// Mitsubishi GX Works2 project: PLC (21)   PLC: FX3G
// PLC

// global labels: Global1
VAR_GLOBAL
  light1 AT Y010 : BOOL;
  EmergencySwitch AT X007 : BOOL;
  OrangeReg AT D1100 : REAL;  (* STARTDAY *)
  TangerineReg AT D1105 : REAL;  (* STARTDAY *)
  PomelaReg AT D1110 : REAL;  (* STARTDAY *)
  OrangeCont AT D1115 : REAL;
  TangerineCont AT D1120 : REAL;
  PomelaCont AT D1125 : REAL;
  startSwitch AT X010 : BOOL;  (* STARTDAY *)
  light2 AT M0 : BOOL;  (* STARTDAY *)
END_VAR
VAR_GLOBAL CONSTANT
  two : REAL := 2;
END_VAR
VAR_GLOBAL
  light3 AT M1 : BOOL;  (* STARTDAY *)
  washSwitch AT X002 : BOOL;
  washTimer AT TC1 : BOOL;
END_VAR
VAR_GLOBAL CONSTANT
  three : INT := 30;
END_VAR
VAR_GLOBAL
  washing AT TS1 : BOOL;
  washLight AT Y005 : BOOL;
END_VAR
VAR_GLOBAL CONSTANT
  countTo3 : INT := 30;  (* שלוש שניות *)
  hundred : REAL := 100;
END_VAR
VAR_GLOBAL
  OrangeWashReg AT D1130 : REAL;
  light4 AT M2 : BOOL;  (* אם יש מעל 100 קג תפוזים *)
END_VAR
VAR_GLOBAL CONSTANT
  zeroConst : REAL;
END_VAR
VAR_GLOBAL
  light5 AT M3 : BOOL;  (* אם יש מתחת ל100 קג תפוזים *)
  light6 AT M4 : BOOL;  (* תפוזים נשטפו *)
END_VAR
VAR_GLOBAL CONSTANT
  half : REAL := 0.5;
END_VAR
VAR_GLOBAL
  PomelaWashReg AT D1135 : REAL;
  TangerineWashReg AT D1140 : REAL;
  light7 AT M5 : BOOL;  (* הכל נשטף *)
  squeezeSwitch AT X001 : BOOL;  (* stage 2 start *)
  squeezeCont AT D1145 : REAL;  (* מיכל סחיטה של כלל הפירות *)
  stage2light AT Y001 : BOOL;
  stage3Switch AT X011 : BOOL;
  stage3Counter AT CC0 : BOOL;
END_VAR
VAR_GLOBAL CONSTANT
  countTo2 : INT := 2;  (* שתי לחיצות *)
END_VAR
VAR_GLOBAL
  stage3Start AT CS0 : BOOL;
  light8 AT M6 : BOOL;
END_VAR
VAR_GLOBAL CONSTANT
  halfSec : INT := 5;
END_VAR
VAR_GLOBAL
  squeezeTimer AT TC2 : BOOL;
  flashing AT TS2 : BOOL;
  flashlight2 AT Y002 : BOOL;
  squeezeTimer2 AT TC3 : BOOL;
  flashlight3 AT Y003 : BOOL;
  flashing2 AT TS3 : BOOL;
  stage3TotalTime AT TC4 : BOOL;
  threeSecOff AT TS4 : BOOL;  (* כיבוי אורות מהבהבים לאחר 3 שניות *)
  light9 AT M7 : BOOL;  (* תהליך הסחיטה הסתיים *)
  juiceCont AT D1150 : REAL;  (* מיכל מיץ סחוט *)
  light10 AT M8 : BOOL;
  analog2 AT D8281 : WORD;
  analogOutput2 AT D1160 : WORD;
END_VAR
VAR_GLOBAL CONSTANT
  fourHundred : REAL := 400.0;
END_VAR
VAR_GLOBAL
  qualityCheckReg AT D1155 : REAL;
END_VAR
VAR_GLOBAL CONSTANT
  One : REAL := 1.0;
  five : REAL := 5.0;
END_VAR
VAR_GLOBAL
  light11 AT M9 : BOOL;
  light12 AT M10 : BOOL;
  qualityIsGood AT Y004 : BOOL;
  qualityIsAmazing AT Y004 : BOOL;
END_VAR
VAR_GLOBAL CONSTANT
  countTo5 : INT := 50;
END_VAR
VAR_GLOBAL
  qualityTimer AT TC5 : BOOL;
  TS05 AT TS5 : BOOL;
  light13 AT M11 : BOOL;
  failCounter AT CC1 : BOOL;
  disgustingJuice AT CS1 : BOOL;  (* נכשל פעמיים בבדיקת איכות *)
  PerfectJuiceStorage AT D1165 : REAL;
  stage4Switch AT X003 : BOOL;
  light14 AT M12 : BOOL;
  light15 AT M13 : BOOL;
  light16 AT M14 : BOOL;
  repairMachine AT X006 : BOOL;  (* התקשרות לטכנאי לתיקון *)
  maxFruitReg AT D1170 : REAL;
  analogOutput AT D8282 : WORD;
  endOfDay AT M15 : BOOL;
  repairTimer AT TC6 : BOOL;  (* זמן תיקון *)
  repairFlash AT TC7 : BOOL;
  repairLight AT Y006 : BOOL;
  light17 AT M16 : BOOL;
  repairFlashING AT TS7 : BOOL;
  repairFakeFlash AT TC8 : BOOL;
  light18 AT M17 : BOOL;
  repairSchedule AT TS8 : BOOL;
  light19 AT M18 : BOOL;
  endOfIteration AT M19 : BOOL;  (* סוף איטרציה *)
  howLongRepair AT D1175 : WORD;
END_VAR

// task Task_01 (event TRUE, interval 0, priority 31): POU_01

PROGRAM POU_01
(* structured ladder/FBD written out as ST: instructions are called as NAME(EN, inputs, outputs); _pN, _eN, _tN stand for wires *)
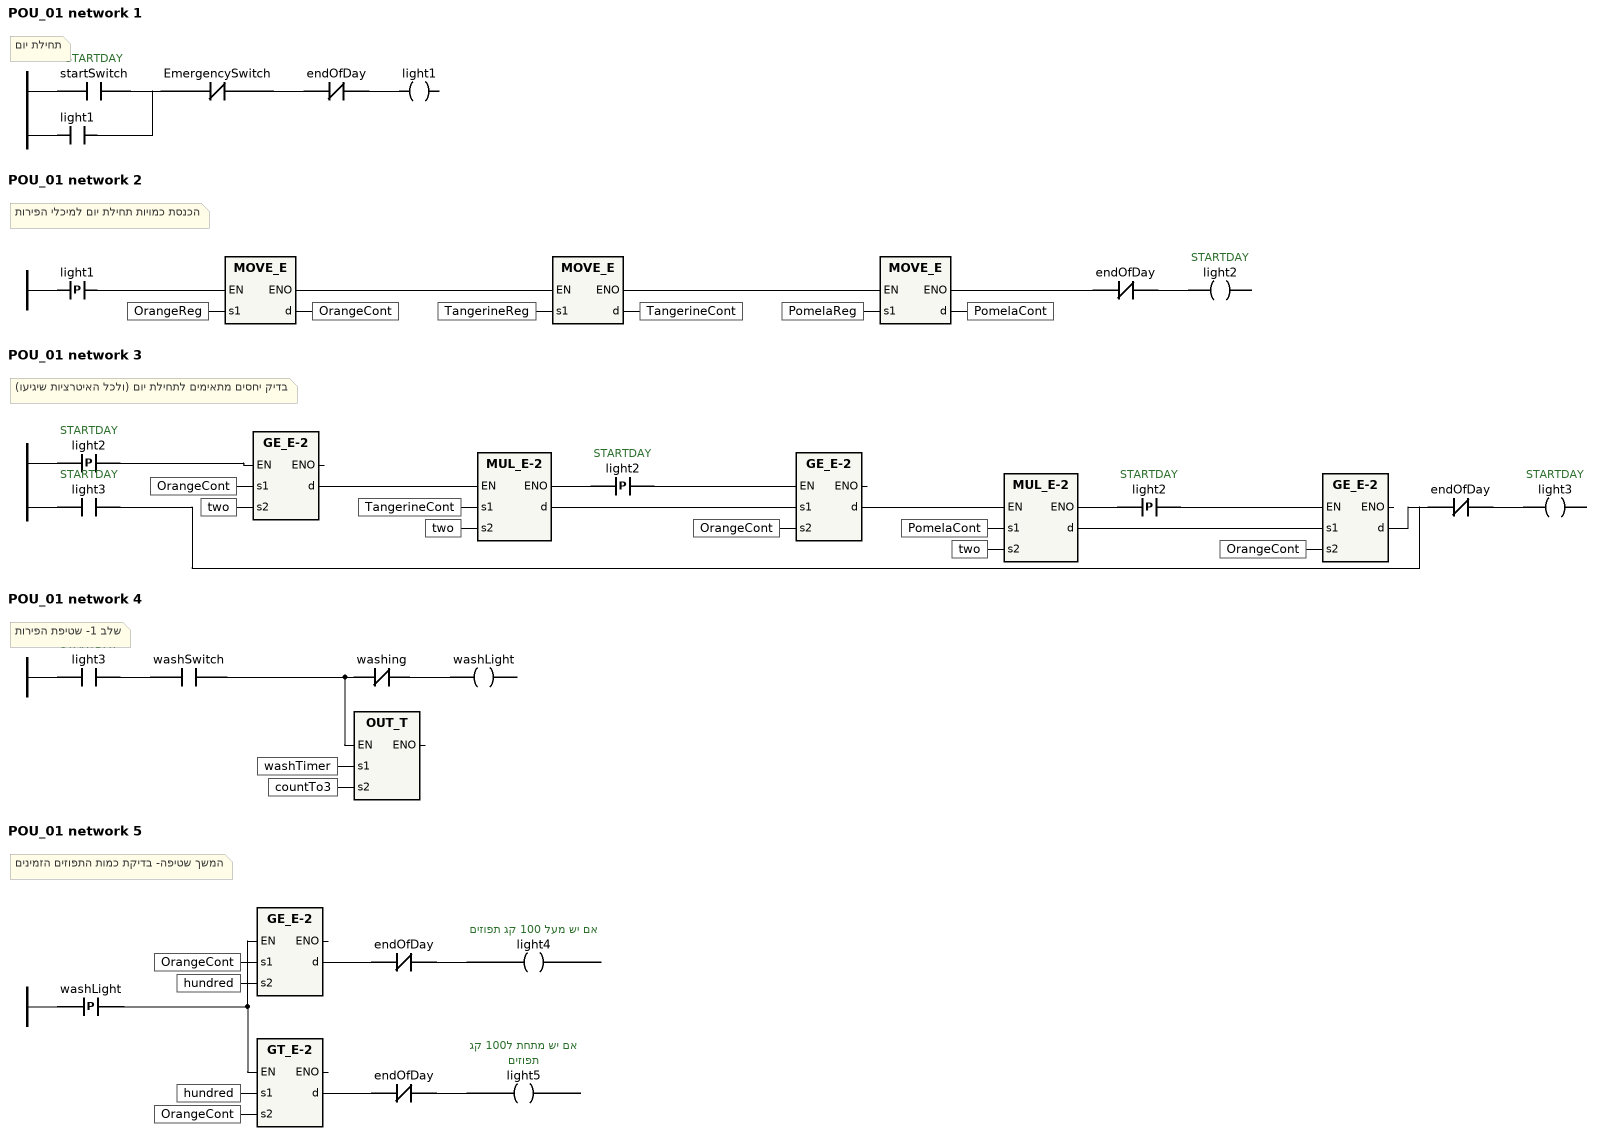
(* network 1 *)
(* תחילת יום *)
light1 := ((startSwitch OR light1) AND NOT EmergencySwitch) AND NOT endOfDay;
(* network 2 *)
(* הכנסת כמויות תחילת יום למיכלי הפירות *)
_e1 := MOVE_E(LDP(TRUE, light1), OrangeReg, OrangeCont);
_e2 := MOVE_E(_e1, TangerineReg, TangerineCont);
_e3 := MOVE_E(_e2, PomelaReg, PomelaCont);
light2 := _e3 AND NOT endOfDay;
(* network 3 *)
(* בדיק יחסים מתאימים לתחילת יום (ולכל האיטרציות שיגיעו) *)
GE_E(LDP(TRUE, light2), OrangeCont, two, _t1);
_e3 := MUL_E(_t1, TangerineCont, two, _t2);
GE_E(_e3 AND LDP(TRUE, light2), _t2, OrangeCont, _t4);
_e6 := MUL_E(_t4, PomelaCont, two, _t5);
GE_E(_e6 AND LDP(TRUE, light2), _t5, OrangeCont, _t7);
light3 := (_t7 OR light3) AND NOT endOfDay;
(* network 4 *)
(* שלב 1- שטיפת הפירות *)
_p1 := light3 AND washSwitch;
washLight := _p1 AND NOT washing;
OUT_T(_p1, washTimer, countTo3);
(* network 5 *)
(* המשך שטיפה- בדיקת כמות התפוזים הזמינים *)
_p1 := LDP(TRUE, washLight);
GE_E(_p1, OrangeCont, hundred, _t2);
light4 := _t2 AND NOT endOfDay;
GT_E(_p1, hundred, OrangeCont, _t3);
light5 := _t3 AND NOT endOfDay;
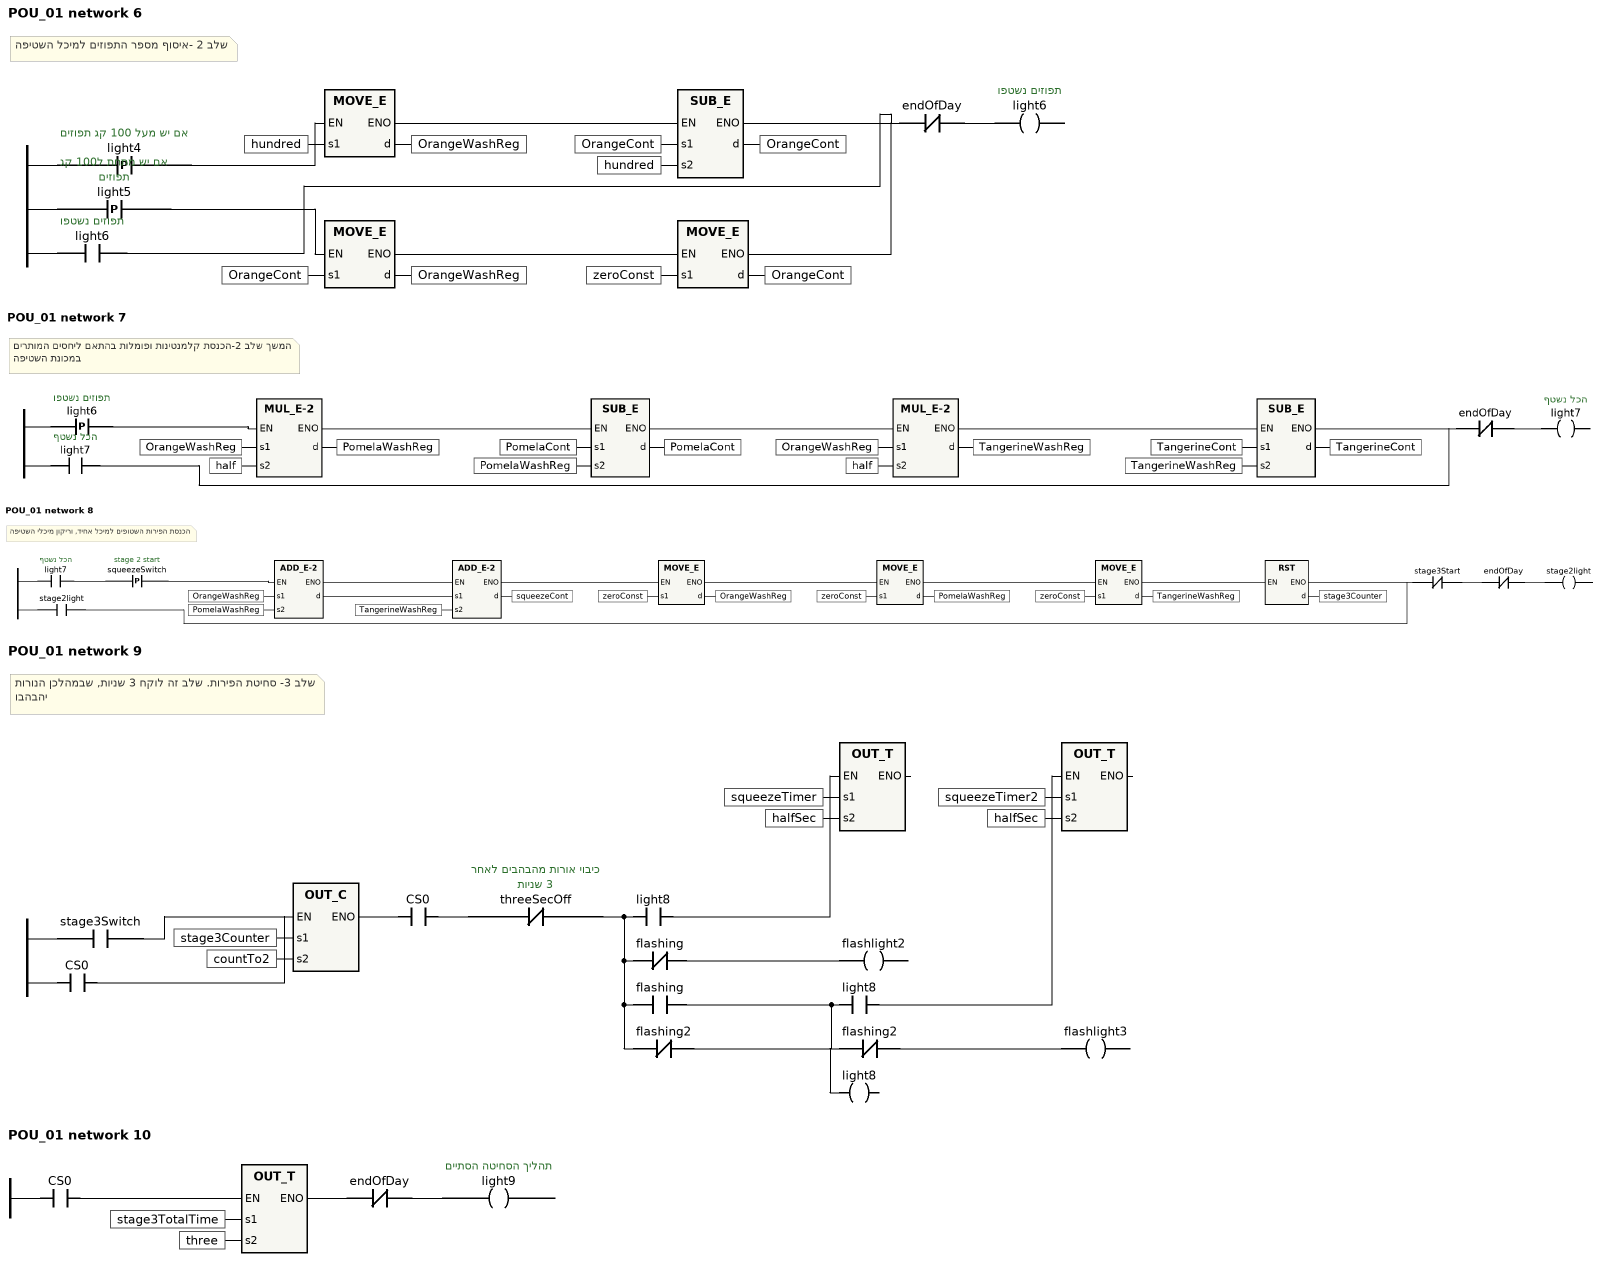
(* network 6 *)
(* שלב 2 -איסוף מספר התפוזים למיכל השטיפה *)
_e1 := MOVE_E(LDP(TRUE, light4), hundred, OrangeWashReg);
_e2 := SUB_E(_e1, OrangeCont, hundred, OrangeCont);
_e3 := MOVE_E(LDP(TRUE, light5), OrangeCont, OrangeWashReg);
_e4 := MOVE_E(_e3, zeroConst, OrangeCont);
light6 := (_e2 OR _e4 OR light6) AND NOT endOfDay;
(* network 7 *)
(* המשך שלב 2-הכנסת קלמנטינות ופומלות בהתאם ליחסים המותרים במכונת השטיפה *)
_e1 := MUL_E(LDP(TRUE, light6), OrangeWashReg, half, PomelaWashReg);
_e2 := SUB_E(_e1, PomelaCont, PomelaWashReg, PomelaCont);
_e3 := MUL_E(_e2, OrangeWashReg, half, TangerineWashReg);
_e4 := SUB_E(_e3, TangerineCont, TangerineWashReg, TangerineCont);
light7 := (_e4 OR light7) AND NOT endOfDay;
(* network 8 *)
(* הכנסת הפירות השטופים למיכל אחיד, וריקון מיכלי השטיפה *)
_e2 := ADD_E(light7 AND LDP(TRUE, squeezeSwitch), OrangeWashReg, PomelaWashReg, _t1);
_e3 := ADD_E(_e2, _t1, TangerineWashReg, squeezeCont);
_e4 := MOVE_E(_e3, zeroConst, OrangeWashReg);
_e5 := MOVE_E(_e4, zeroConst, PomelaWashReg);
_e6 := MOVE_E(_e5, zeroConst, TangerineWashReg);
_e7 := RST(_e6, stage3Counter);
stage2light := ((_e7 OR stage2light) AND NOT stage3Start) AND NOT endOfDay;
(* network 9 *)
(* שלב 3- סחיטת הפירות. שלב זה לוקח 3 שניות, שבמהלכן הנורות יהבהבו *)
_e1 := OUT_C(stage3Switch OR CS0, stage3Counter, countTo2);
_p2 := _e1 AND CS0 AND NOT threeSecOff;
OUT_T(_p2 AND light8, squeezeTimer, halfSec);
flashlight2 := _p2 AND NOT flashing;
_p3 := _p2 AND flashing;
OUT_T(_p3 AND light8, squeezeTimer2, halfSec);
flashlight3 := _p3 AND NOT flashing2;
light8 := _p2 AND NOT flashing2;
(* network 10 *)
_e1 := OUT_T(CS0, stage3TotalTime, three);
light9 := _e1 AND NOT endOfDay;
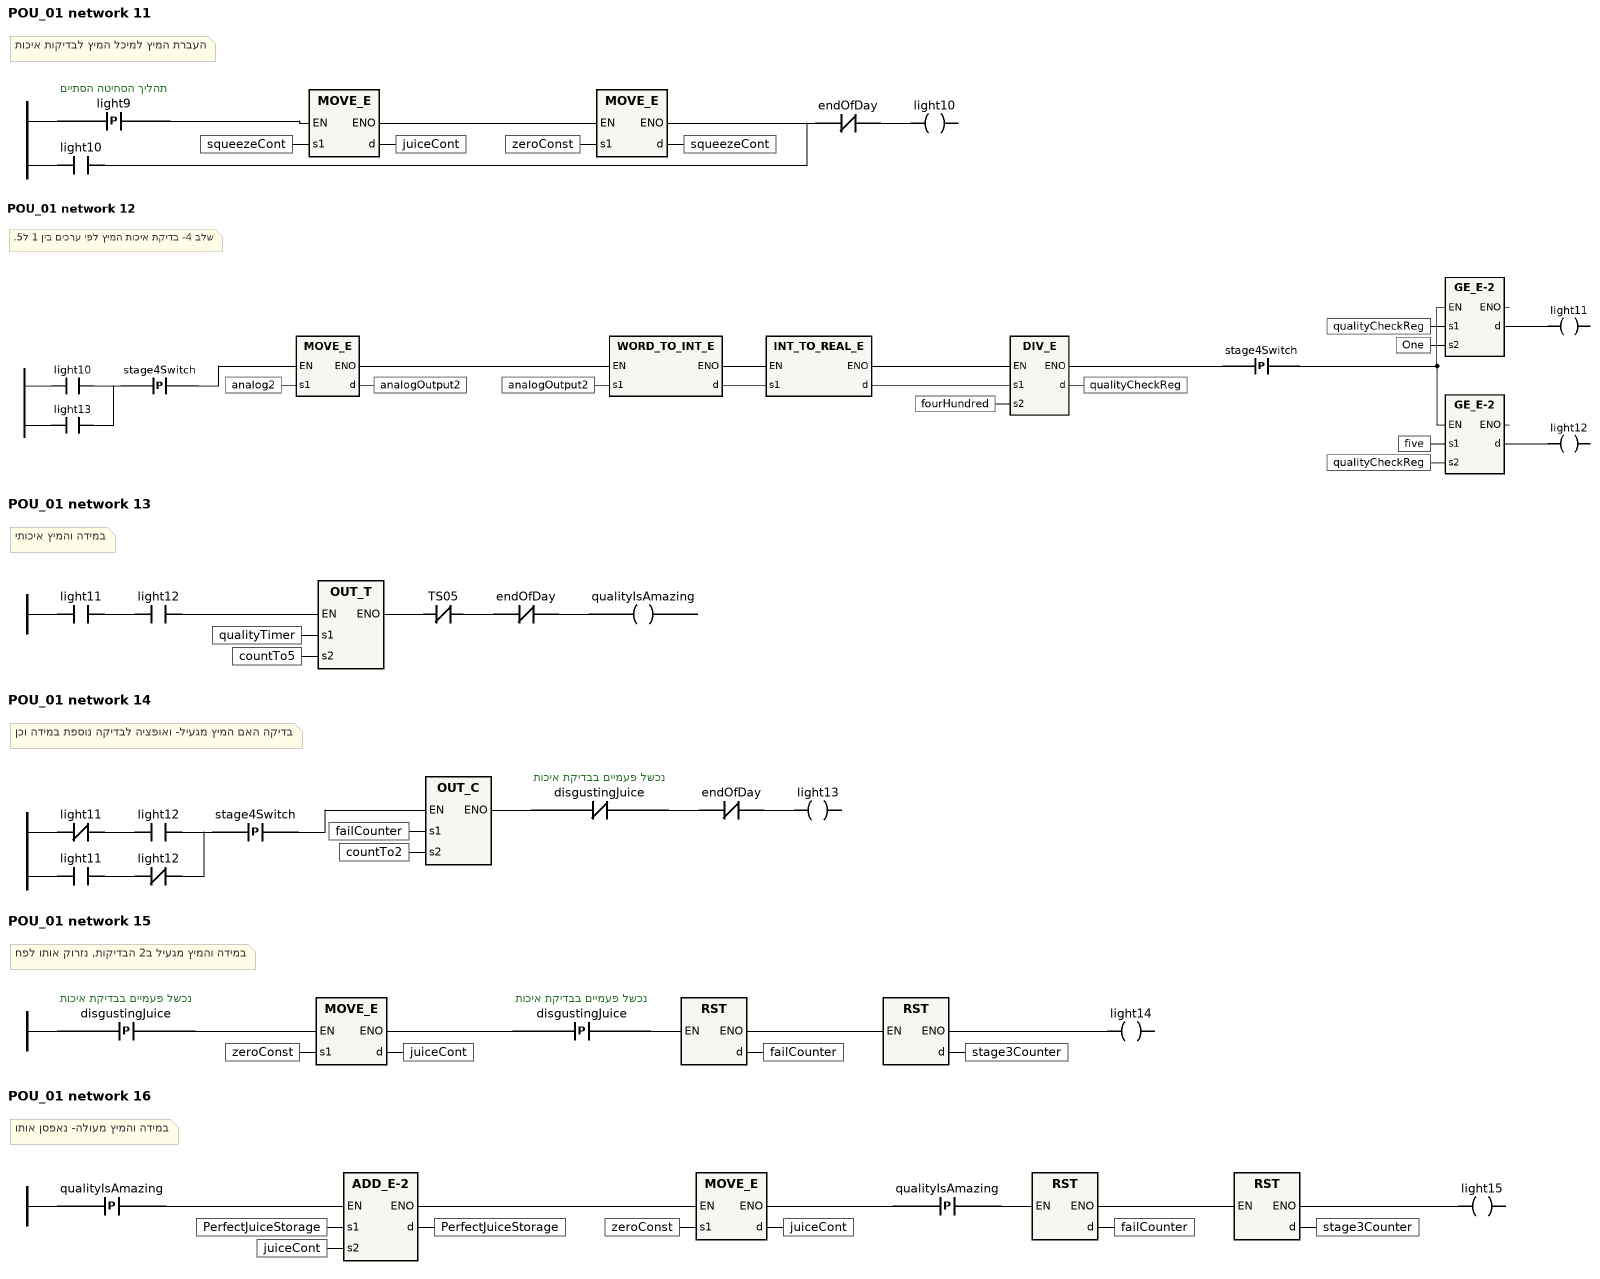
(* network 11 *)
(* העברת המיץ למיכל המיץ לבדיקות איכות *)
_e1 := MOVE_E(LDP(TRUE, light9), squeezeCont, juiceCont);
_e2 := MOVE_E(_e1, zeroConst, squeezeCont);
light10 := (_e2 OR light10) AND NOT endOfDay;
(* network 12 *)
(* שלב 4- בדיקת איכות המיץ לפי ערכים בין 1 ל5. *)
_e1 := MOVE_E((light10 OR light13) AND LDP(TRUE, stage4Switch), analog2, analogOutput2);
_e3 := WORD_TO_INT_E(_e1, analogOutput2, _t2);
_e5 := INT_TO_REAL_E(_e3, _t2, _t4);
_e6 := DIV_E(_e5, _t4, fourHundred, qualityCheckReg);
_p7 := _e6 AND LDP(TRUE, stage4Switch);
GE_E(_p7, qualityCheckReg, One, _t8);
light11 := _t8;
GE_E(_p7, five, qualityCheckReg, _t9);
light12 := _t9;
(* network 13 *)
(* במידה והמיץ איכותי *)
_e1 := OUT_T(light11 AND light12, qualityTimer, countTo5);
qualityIsAmazing := _e1 AND NOT TS05 AND NOT endOfDay;
(* network 14 *)
(* בדיקה האם המיץ מגעיל- ואופציה לבדיקה נוספת במידה וכן *)
_e1 := OUT_C(((NOT light11 AND light12) OR (light11 AND NOT light12)) AND LDP(TRUE, stage4Switch), failCounter, countTo2);
light13 := _e1 AND NOT disgustingJuice AND NOT endOfDay;
(* network 15 *)
(* במידה והמיץ מגעיל ב2 הבדיקות, נזרוק אותו לפח *)
_e1 := MOVE_E(LDP(TRUE, disgustingJuice), zeroConst, juiceCont);
_e2 := RST(_e1 AND LDP(TRUE, disgustingJuice), failCounter);
_e3 := RST(_e2, stage3Counter);
light14 := _e3;
(* network 16 *)
(* במידה והמיץ מעולה- נאפסן אותו *)
_e1 := ADD_E(LDP(TRUE, qualityIsAmazing), PerfectJuiceStorage, juiceCont, PerfectJuiceStorage);
_e2 := MOVE_E(_e1, zeroConst, juiceCont);
_e3 := RST(_e2 AND LDP(TRUE, qualityIsAmazing), failCounter);
_e4 := RST(_e3, stage3Counter);
light15 := _e4;
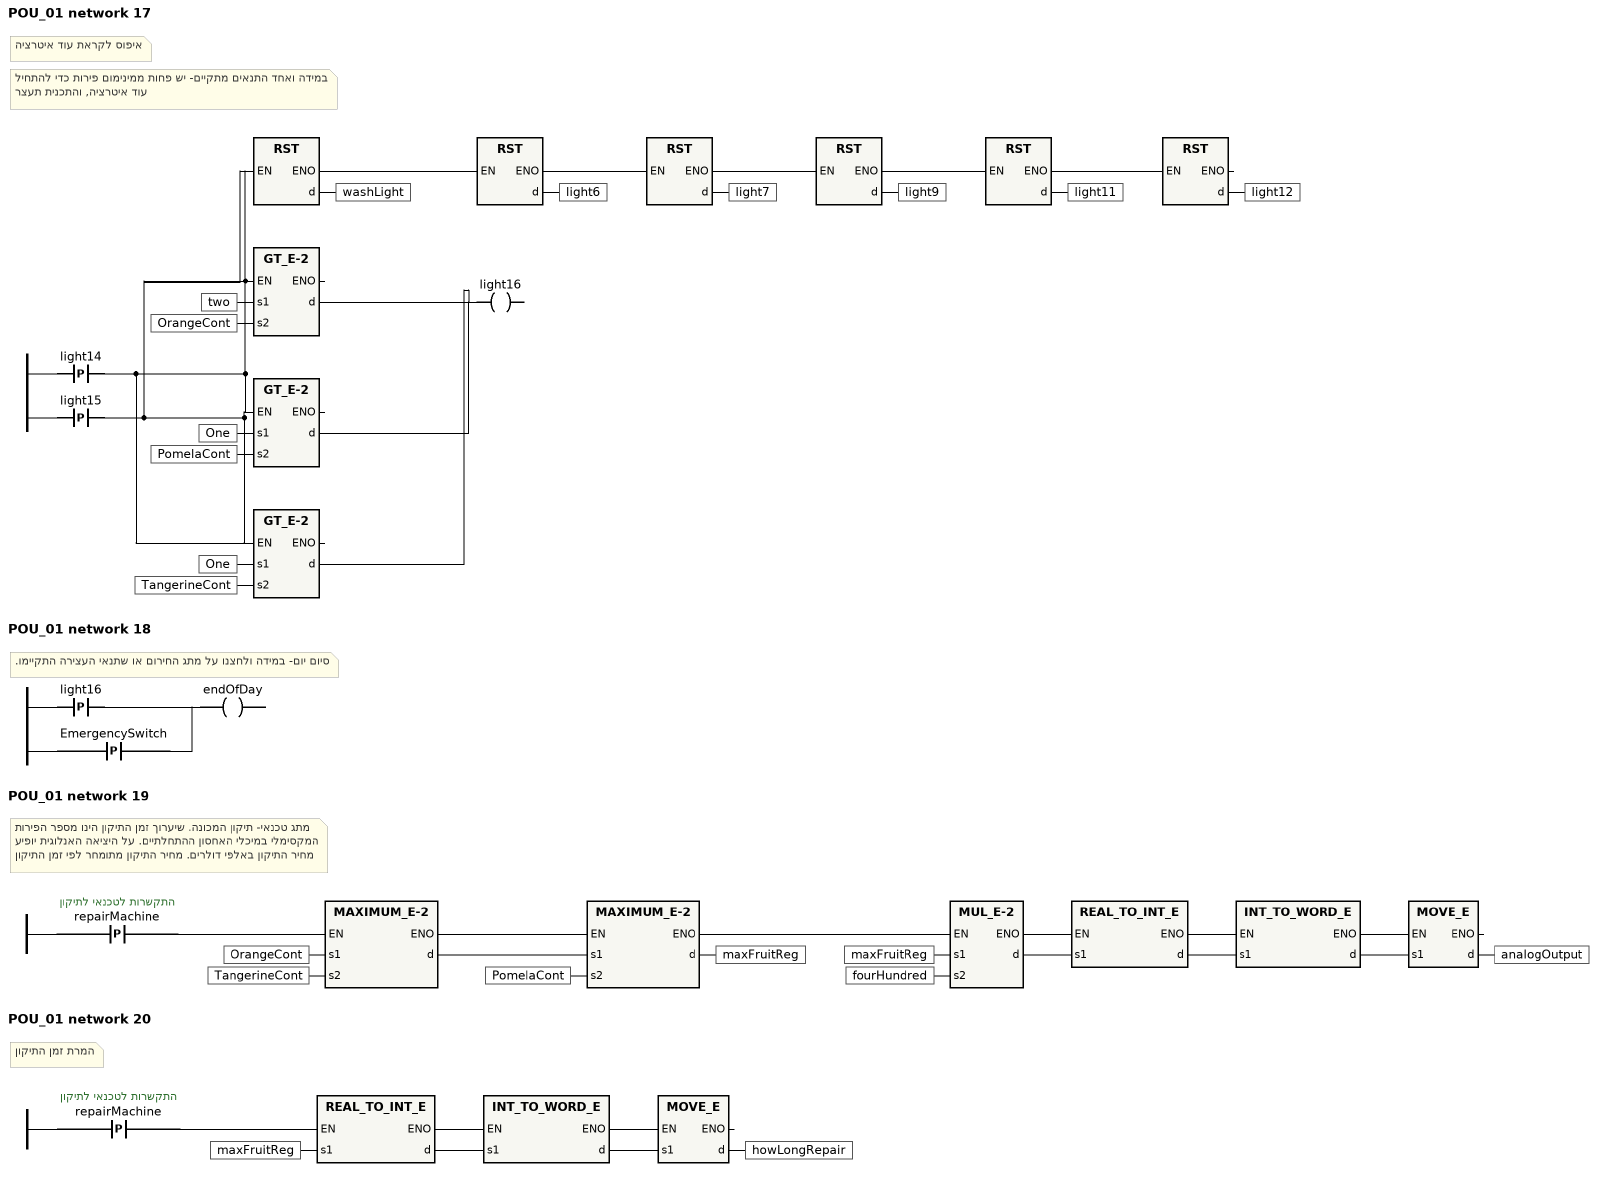
(* network 17 *)
(* איפוס לקראת עוד איטרציה *)
(* במידה ואחד התנאים מתקיים- יש פחות ממינימום פירות כדי להתחיל עוד איטרציה, והתכנית תעצר *)
_p1 := LDP(TRUE, light14) OR LDP(TRUE, light15);
_e2 := RST(_p1, washLight);
_e3 := RST(_e2, light6);
_e4 := RST(_e3, light7);
_e5 := RST(_e4, light9);
_e6 := RST(_e5, light11);
RST(_e6, light12);
GT_E(_p1, two, OrangeCont, _t7);
GT_E(_p1, One, PomelaCont, _t8);
GT_E(_p1, One, TangerineCont, _t9);
light16 := _t7 OR _t8 OR _t9;
(* network 18 *)
(* סיום יום- במידה ולחצנו על מתג החירום או שתנאי העצירה התקיימו. *)
endOfDay := LDP(TRUE, light16) OR LDP(TRUE, EmergencySwitch);
(* network 19 *)
(* מתג טכנאי- תיקון המכונה. שיערוך זמן התיקון הינו מספר הפירות המקסימלי במיכלי האחסון ההתחלתיים. על היציאה האנלוגית יופיע מחיר התיקון באלפי דולרים. מחיר התיקון מתומחר לפי זמן התיקון *)
_e2 := MAXIMUM_E(LDP(TRUE, repairMachine), OrangeCont, TangerineCont, _t1);
_e3 := MAXIMUM_E(_e2, _t1, PomelaCont, maxFruitReg);
_e5 := MUL_E(_e3, maxFruitReg, fourHundred, _t4);
_e7 := REAL_TO_INT_E(_e5, _t4, _t6);
_e9 := INT_TO_WORD_E(_e7, _t6, _t8);
MOVE_E(_e9, _t8, analogOutput);
(* network 20 *)
(* המרת זמן התיקון *)
_e2 := REAL_TO_INT_E(LDP(TRUE, repairMachine), maxFruitReg, _t1);
_e4 := INT_TO_WORD_E(_e2, _t1, _t3);
MOVE_E(_e4, _t3, howLongRepair);
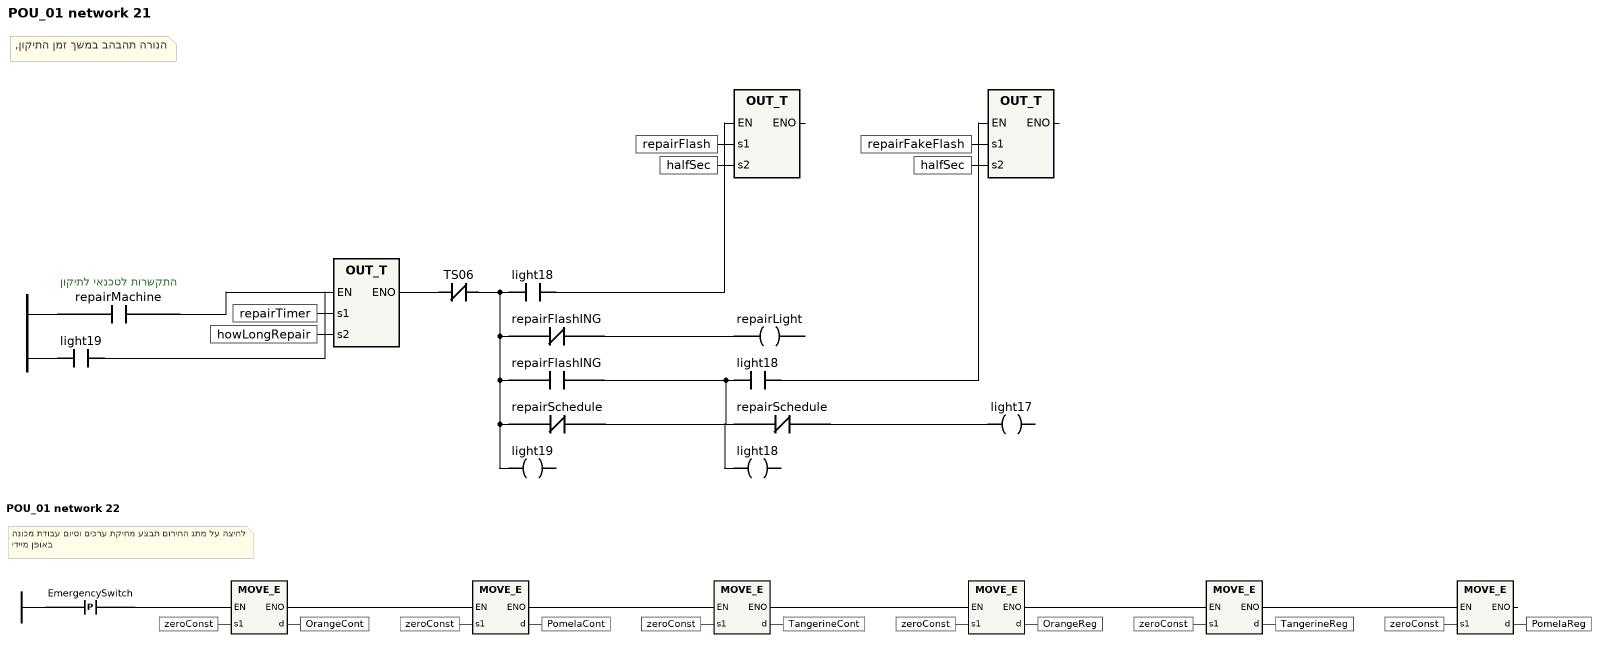
(* network 21 *)
(* הנורה תהבהב במשך זמן התיקון, *)
_e1 := OUT_T(repairMachine OR light19, repairTimer, howLongRepair);
_p2 := _e1 AND NOT TS06;
OUT_T(_p2 AND light18, repairFlash, halfSec);
repairLight := _p2 AND NOT repairFlashING;
_p3 := _p2 AND repairFlashING;
OUT_T(_p3 AND light18, repairFakeFlash, halfSec);
light17 := _p3 AND NOT repairSchedule;
light18 := _p2 AND NOT repairSchedule;
light19 := _p2;
(* network 22 *)
(* לחיצה על מתג החירום תבצע מחיקת ערכים וסיום עבודת מכונה באופן מיידי *)
_e1 := MOVE_E(LDP(TRUE, EmergencySwitch), zeroConst, OrangeCont);
_e2 := MOVE_E(_e1, zeroConst, PomelaCont);
_e3 := MOVE_E(_e2, zeroConst, TangerineCont);
_e4 := MOVE_E(_e3, zeroConst, OrangeReg);
_e5 := MOVE_E(_e4, zeroConst, TangerineReg);
MOVE_E(_e5, zeroConst, PomelaReg);
END_PROGRAM
